(* PLC project b22, MITSUBISHI ELECTRIC CORPORATION GX Works3 1.120A *)
(* stored: companyURL http://www.mitsubishielectric.com, creationDateTime 2026-10-05T05:48:24+07:00, modificationDateTime 2026-06-25T03:20:25+07:00 *)

PROGRAM Timer

(* LD diagram, written out as Structured Text *)
END_PROGRAM

PROGRAM Auto

(* LD diagram, written out as Structured Text *)
END_PROGRAM

PROGRAM output

(* LD diagram, written out as Structured Text *)
END_PROGRAM

CONFIGURATION 
  RESOURCE MAIN ON PLC
    PROGRAM Timer : Timer;
    PROGRAM Auto : Auto;
    PROGRAM output : output;
  END_RESOURCE
END_CONFIGURATION
